{attribute 'pack_mode' := '1'}
TYPE ST_MoveToStationDataIn :
STRUCT
	eInputType					: UINT;										(* The vehicle/vehicles that will be moved. *)
	sInput						: STRING(30);								(* Depending on the input type, the input can be the ID of a vehicle, last, article, last type, cell or station. *)
	sStationID					: STRING(30);								(* The ID of the station that will be moved to. *)
	eDirection					: BYTE;										(* 0: BiDirectional, 1: Forward, 2: Backward *)
	nFollowID					: UINT := 0;
	fVelocity					: REAL;
	fAcceleration				: REAL;
END_STRUCT
END_TYPE

(* stored: Version 1.1.0.1, ProductVersion 3.1.4024.5
   DUT ST_MoveToStationDataIn: Id {2117ffdc-ba38-4257-a0fe-48d03e7069e3} *)
